// Mitsubishi GX Works2 project: pisca pisca   PLC: Q03UDV

PROGRAM MAIN
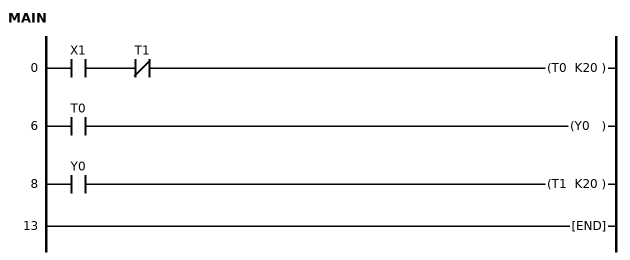
0     LD      X1
      ANI     T1
      OUT     T0 K20
6     LD      T0
      OUT     Y0
8     LD      Y0
      OUT     T1 K20
13    END
END_PROGRAM
